// TwinCAT 3 PLC project Demo
// libraries:
//   DemoLib, * (Demo)
//   Tc2_EtherCAT, * (Beckhoff Automation GmbH)
//   Tc2_Standard, * (Beckhoff Automation GmbH)
//   Tc2_System, * (Beckhoff Automation GmbH)
//   Tc2_SerialCom, * (Beckhoff Automation GmbH)
//   Tc2_Missing, * (Nobody)
// project tree:
//   GVLs/ GVL_Main.TcGVL, GVL_Quoted.TcGVL
//   DUTs/ ST_Point.TcDUT, E_Mode.TcDUT
//   POUs/ MAIN.TcPOU, FB_Motor.TcPOU, I_Motor.TcIO (not stored), F_Add.TcPOU
//   / PlcTask.TcTTO
//   Visu/ Screen.TcVIS (not stored)
// real-time tasks:
//   TASK PlcTask: cycle T#1ms, priority 20, ADS port 350

CONFIGURATION Demo
    RESOURCE PLC ON TwinCAT3
        TASK PlcTask(INTERVAL := T#1ms, PRIORITY := 20);
        PROGRAM MAIN WITH PlcTask : MAIN;
    END_RESOURCE
END_CONFIGURATION

// ---- DUTs/ST_Point.TcDUT
TYPE ST_Point :
STRUCT
	x : INT;
	y : INT;
END_STRUCT
END_TYPE

// ---- DUTs/E_Mode.TcDUT
{attribute 'qualified_only'}
TYPE E_Mode :
(
	Idle := 0,
	Run := 1
) INT;
END_TYPE

// ---- GVLs/GVL_Main.TcGVL
{attribute 'qualified_only'}
VAR_GLOBAL
	counter : DINT;
	origin : ST_Point;
	mode : E_Mode := E_Mode.Idle;
END_VAR

// ---- GVLs/GVL_Quoted.TcGVL
{attribute "qualified_only"}
VAR_GLOBAL
	quotedFlag : BOOL;
END_VAR

// ---- POUs/MAIN.TcPOU
PROGRAM MAIN
VAR
	fbMotor : FB_Motor;
	pt : ST_Point;
	sum : INT;
	spd : INT;
	ok : BOOL;
	lib : FB_LibThing;
	ecState : FB_EcGetSlaveState;
	addr : UINT;
END_VAR

GVL_Main.counter := GVL_Main.counter + 1;
fbMotor.enable := GVL_Main.mode = E_Mode.Run;
fbMotor();
spd := fbMotor.Speed;
ok := fbMotor.Start(force := FALSE);
pt := GVL_Main.origin;
sum := F_Add(a := pt.x, b := pt.y);
lib(execute := ok);
ecState(sNetId := '', nSlaveAddr := addr, bExecute := ok);
quotedFlag := ecState.bBusy;

END_PROGRAM

// ---- POUs/FB_Motor.TcPOU
{attribute 'reflection'}
(* A small motor block with methods, an action and a property. *)
FUNCTION_BLOCK FB_Motor
VAR_INPUT
	enable : BOOL;
END_VAR
VAR_OUTPUT
	running : BOOL;
END_VAR
VAR
	speedSet : INT;
	startCount : DINT;
END_VAR

running := enable;
IF NOT running THEN
	speedSet := 0;
END_IF

METHOD PUBLIC Start : BOOL
VAR_INPUT
	force : BOOL;
END_VAR
startCount := startCount + 1;
Start := enable OR force;
END_METHOD

ACTION Reset:
running := FALSE;
startCount := 0;
END_ACTION

PROPERTY PUBLIC Speed : INT
GET
Speed := speedSet;
END_GET
SET
speedSet := Speed;
END_SET
END_PROPERTY

METHOD Stop
VAR
	wasRunning : BOOL;
END_VAR
wasRunning := running;
running := FALSE;
END_METHOD

END_FUNCTION_BLOCK

// ---- POUs/F_Add.TcPOU
FUNCTION F_Add : INT
VAR_INPUT
	a : INT;
	b : INT;
END_VAR

F_Add := a + b;

END_FUNCTION
